Universal Robots PolyScope program: test_socket_new.urp

Program test_socket_new (installation=default directory=/home/ur/ursim-current/programs createdIn=5.9.4.1031232 lastSavedIn=5.9.4.1031232 robotSerialNumber=20195399999)
Calibrated DH parameters: a=[0, -0.24355, -0.2132, 0, 0, 0]; d=[0.15185, 0, 0, 0.13105, 0.08535, 0.0921]; alpha=[1.570796, 0, 0, 1.570796, -1.570796, 0]; deltaTheta=[0, 0, 0, 0, 0, 0]
BeforeStart
  Loop While (checkContinuously=false) expression=not socket_open("192.168.2.130",50002)
    Wait Sleep waitTime=0.05
  data := socket_read_ascii_float(6)
  If to_str(data[1])≟"nan"
    Script: socket_close()
    Halt
  desired_q := [data[1], data[2], data[3], data[4], data[5], data[6]]
  MoveJ speed 30 deg/s, acceleration 40 deg/s^2 (useActiveTCP=true) feature=Base
    Waypoint Waypoint (Variable): variable=desired_q
  Wait Sleep waitTime=0.5
  current_p := get_actual_tcp_pose()
  desired_p := get_forward_kin(desired_q)
  If point_distance(current_p, desired_p) > 0.01
    Script: socket_send_string("Posicion no alcanzada")
    Script: socket_close()
    Halt
  Script: socket_send_string("Ready")
  Wait Sleep waitTime=0.05
Robot Program (runOnlyOnce=false)
  data := socket_read_ascii_float(6)
  Script: socket_send_string(get_actual_joint_positions())
  If to_str(data[1])≟"nan"
    Script: socket_close()
    Halt
  desired_q := [data[1], data[2], data[3], data[4], data[5], data[6]]
Thread Thread_1 (runOnlyOnce=false)
  current_p := get_actual_tcp_pose()
  desired_p := get_forward_kin(desired_q)
  If point_distance(current_p, desired_p) < 0.01
    Script: servoj(desired_q,0,0,0.008,0.1,150)
  Else 
    Script: servoj(desired_q,0,0,0.008,0.5,100)
